INTERFACE I_Cam_Ctrl

END_INTERFACE

(* stored: Version 1.1.0.1, ProductVersion 3.1.4024.12
   Itf I_Cam_Ctrl: Id {d121444c-d264-002c-3692-487f8a771313} *)
